FUNCTION_BLOCK FB_AxisRead5042
VAR_INPUT
	bExecute: BOOL;
	bReset: BOOL;
	stDriveRef: ST_DriveRef;
END_VAR
VAR_IN_OUT
	stConfig: ST_AxisParams;
	Axis: AXIS_REF;
END_VAR
VAR_OUTPUT
	bBusy: BOOL;
	bError: BOOL;
	iAdsErrId: UINT;
	iCANopenErrId: UINT;
END_VAR
VAR
	iCycles: INT := 0;
	bReadOk: BOOL := FALSE;
	bInnerExec: BOOL := FALSE;
	fbReadEncSupply: FB_CoERead_ByDriveRef;
	nIndEncSupply: WORD;
	fbReadEncClock: FB_CoERead_ByDriveRef;
	nIndEncClock: WORD;
	fbReadEncMultiBits: FB_CoERead_ByDriveRef;
	nIndEncMultiBits: WORD;
	fbReadEncSingleBits: FB_CoERead_ByDriveRef;
	nIndEncSingleBits: WORD;
END_VAR

// File auto-generated! Take care editing!
// Clears errors and allows a new read
IF bReset THEN
	bExecute := FALSE;
	bReset := FALSE;
END_IF
// Fails in the first n cycles depending on terminals, wait a bit
IF NOT bReadOk THEN
	iCycles := iCycles + 1;
	IF iCycles > 100 THEN
		bReadOk := TRUE;
	END_IF
END_IF
bInnerExec := bExecute AND bReadOk;
nIndEncSupply := 16#8008;
fbReadEncSupply(bExecute:=bInnerExec,
	stDriveRef:=stDriveRef,
	nindex:=nIndEncSupply,
	nSubIndex:=12,
	pDstBuf:=ADR(stConfig.enc_supply),
	cbBufLen:=SIZEOF(stConfig.enc_supply));
CASE stDriveRef.nDriveNo OF
	0:
		nIndEncClock := 16#8008;
	1:
		nIndEncClock := 16#8018;
END_CASE
fbReadEncClock(bExecute:=bInnerExec,
	stDriveRef:=stDriveRef,
	nindex:=nIndEncClock,
	nSubIndex:=13,
	pDstBuf:=ADR(stConfig.enc_clock),
	cbBufLen:=SIZEOF(stConfig.enc_clock));
CASE stDriveRef.nDriveNo OF
	0:
		nIndEncMultiBits := 16#8008;
	1:
		nIndEncMultiBits := 16#8018;
END_CASE
fbReadEncMultiBits(bExecute:=bInnerExec,
	stDriveRef:=stDriveRef,
	nindex:=nIndEncMultiBits,
	nSubIndex:=15,
	pDstBuf:=ADR(stConfig.enc_multi_bits),
	cbBufLen:=SIZEOF(stConfig.enc_multi_bits));
CASE stDriveRef.nDriveNo OF
	0:
		nIndEncSingleBits := 16#8008;
	1:
		nIndEncSingleBits := 16#8018;
END_CASE
fbReadEncSingleBits(bExecute:=bInnerExec,
	stDriveRef:=stDriveRef,
	nindex:=nIndEncSingleBits,
	nSubIndex:=16,
	pDstBuf:=ADR(stConfig.enc_single_bits),
	cbBufLen:=SIZEOF(stConfig.enc_single_bits));

END_FUNCTION_BLOCK

(* stored: Version 1.1.0.1, ProductVersion 3.1.4020.12
   POU FB_AxisRead5042: Id {f8e69a50-2a54-4489-b7d7-965f7b44587e}, SpecialFunc None *)
